// LS Electric XG5000 project: 연습 문제1
// PLC LSPLC
// module base 0 slot 0: 입출력 모듈:XBC-DR14E (DC 24V 입력 8점, 릴레이 출력 6점)

PROGRAM NewProgram (task: 스캔 프로그램)

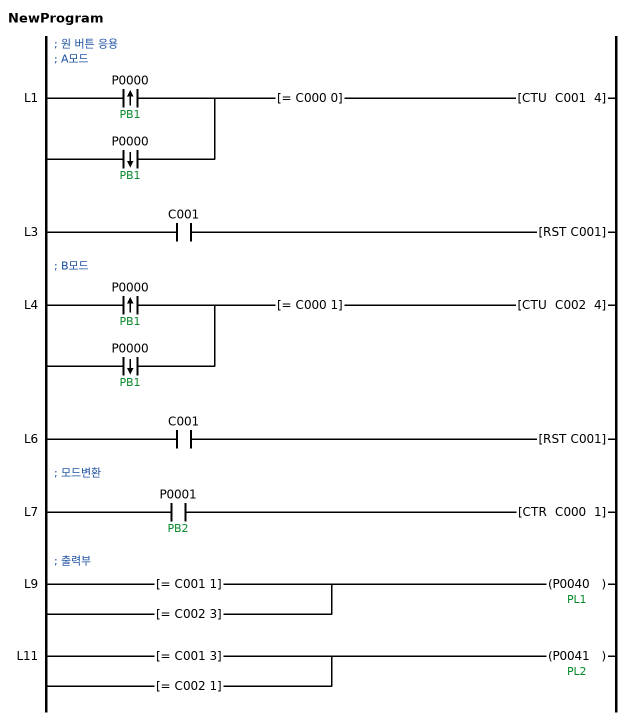
// 원 버튼 응용
; L1
LOADP     P0000	// PB1
ORN       P0000	// PB1
AND=      C000 0
CTU       C001 4
// output comment: A모드
; L3
LOAD      C001
RST       C001
; L4
LOADP     P0000	// PB1
ORN       P0000	// PB1
AND=      C000 1
CTU       C002 4
// output comment: B모드
; L6
LOAD      C001
RST       C001
; L7
LOAD      P0001	// PB2
CTR       C000 1
// output comment: 모드변환
// 출력부
; L9
LOAD=     C001 1
OR=       C002 3
OUT       P0040	// PL1
; L11
LOAD=     C001 3
OR=       C002 1
OUT       P0041	// PL2